FUNCTION_BLOCK ABSTRACT TcoInspectorTests EXTENDS TcoCore._internals_TcoContext
VAR
    _result         : TcoInspectors.eInspectorResult;
    _isOverIspected : BOOL;
    _overallResult  : TcoInspectors.TcoComprehensiveResult;
    _coordinator    : MockCoordinator;
    _retryState     : INT;
END_VAR

METHOD ABSTRACT Inspect : TcoInspectors.IInspector
END_METHOD

METHOD PROTECTED Main
CASE _testId OF
    0:
        _result         := 0;
        _isOverIspected := FALSE;
    eInspectorTests.Inspect:
        THIS^.ProbeDoneWhen(Inspect().UpdateComprehensiveResult(_overallResult).Done);
    eInspectorTests.GetResult:
        _result         := Inspect().Result;
        _isOverIspected := Inspect().OverInspected;
    eInspectorTests.OnFailCarryOn:
        THIS^.ProbeDoneWhen(Inspect().OnFail(_coordinator).CarryOn());
    eInspectorTests.OnFailRetry:
        THIS^.ProbeDoneWhen(Inspect().OnFail(_coordinator).Retry(_retryState));
    eInspectorTests.OnFailTerminate:
        THIS^.ProbeDoneWhen(Inspect().OnFail(_coordinator).Terminate());
END_CASE
END_METHOD

END_FUNCTION_BLOCK

(* stored: Version 1.1.0.1, ProductVersion 3.1.4024.9
   POU TcoInspectorTests: Id {23a7de36-f9c4-0b82-3e65-65f0a2b87059}, SpecialFunc None
   Method Inspect: Id {0a3b37f7-9710-0dae-1c6d-f079d88f81a5}
   Method Main: Id {d3b8a8a4-7806-07ca-3474-7884aa0d6670} *)
